    MS_STOPPING: // ---------------------------------------------------------- STOPPING MOVERS
		(*Movers are coming to a stop here in this state*)

		// Stop all movers
		allMoversHalted				:= TRUE;
		FOR i := 0 TO GVL.NUM_MOVERS - 1 DO
			Mover[i].AxisReference.ReadStatus();
			IF Mover[i].AxisReference.Status.Moving THEN
				allMoversHalted		:= FALSE;
			END_IF
		END_FOR

		GVL.XTS.Cmd.Start			:= FALSE;
 
		IF allMoversHalted THEN
           	GVL.XTS.Sts.State 		:= MS_STOPPED;
		END_IF

    MS_STOPPED: // ------------------------------------------------------------ Stop Command has been sent, hold here
		(*Movers are now stopped, and further Main Commands can be issued to the system*)

        IF GVL.XTS.Cmd.Disable THEN
            GVL.XTS.Cmd.Enable 	:= FALSE;
			GVL.XTS.Cmd.Start	:= FALSE;
            GVL.XTS.Sts.State   := MS_ONESHOT_DISABLE;
        ELSIF GVL.XTS.Cmd.Start THEN
            GVL.XTS.Cmd.Stop 	:= FALSE;
            GVL.XTS.Sts.State   := MS_ENABLING_MOVERS;
        END_IF

        // Unregister everything from everything
        FOR i := 0 TO GVL.NUM_STATIONS - 1 DO	 									Station[i].UnregisterAll();  END_FOR
		FOR i := 0 TO GVL.NUM_MULTISTATIONS - 1 DO									MultiStation[i].UnregisterAll();	END_FOR
//      FOR i := 0 TO SIZEOF(PositionTrigger) / SIZEOF(PositionTrigger[0]) - 1 DO	PositionTrigger[i].UnregisterAll();	END_FOR
//      FOR i := 0 TO SIZEOF(SpeedTrigger) / SIZEOF(SpeedTrigger[0]) - 1 DO 		SpeedTrigger[i].UnregisterAll(); END_FOR
        FOR i := 0 TO SIZEOF(Zone) / SIZEOF(Zone[0]) - 1 DO 						Zone[i].UnregisterAll();	END_FOR

	MS_ONESHOT_DISABLE:	// ------------------------------------------------------- SINGLE CYCLE ISSUE DISABLE COMMANDS
		(*Mover disable commands are issued here, followed by a state tranisition to await completion of the Disabling*)
		FOR i := 0 TO GVL.NUM_MOVERS DO
			Mover[i].Disable();
		END_FOR

		GVL.XTS.Sts.State	:=	MS_DISABLING;

    MS_DISABLING: // --------------------------------------------------- DISABLING MOVERS
		(*Movers are Disabling. During this step, we also Unregister movers from relevant Objectives
		to ensure proper startup behavior*)

        // Unregister everything from everything
        FOR i := 0 TO GVL.NUM_STATIONS - 1 DO	 									Station[i].UnregisterAll();  END_FOR
		FOR i := 0 TO GVL.NUM_MULTISTATIONS - 1 DO									MultiStation[i].UnregisterAll();	END_FOR
//      FOR i := 0 TO SIZEOF(PositionTrigger) / SIZEOF(PositionTrigger[0]) - 1 DO	PositionTrigger[i].UnregisterAll();	END_FOR
//      FOR i := 0 TO SIZEOF(SpeedTrigger) / SIZEOF(SpeedTrigger[0]) - 1 DO 		SpeedTrigger[i].UnregisterAll(); END_FOR
        FOR i := 0 TO SIZEOF(Zone) / SIZEOF(Zone[0]) - 1 DO 						Zone[i].UnregisterAll();	END_FOR
		allMoversDisabled	:= TRUE;

		FOR i := 0 TO gvl.NUM_MOVERS-1 DO
			IF NOT Mover[i].AxisReference.Status.Disabled THEN 
				allMoversDisabled	:= FALSE;
			END_IF
		END_FOR
 
        IF allMoversDisabled THEN
            GVL.XTS.Sts.State		:= MS_DISABLED;
        END_IF

    MS_ERROR: // --------------------------------------------------- ERRORSTATE
		(*A reset command can be included here to clear Mover errors, etc. and return
		to a controlled state*)

    MS_DEBUG: // ------------------------------------------------------- DEV USE ONLY
		(*This state is intentionally left blank, 
		for optional use by a developer during programming*)

END_CASE;

GVL.XTS.Sts.Enabled	:= GVL.XTS.Sts.State = MS_RUN;

// Station Actions
ACT_Orient();
ACT_BallSeat();
ACT_Print();
ACT_Vision();
ACT_Kickout();
ACT_TRAYLOAD();
ACT_IOSim();

ACT_HMIHelper();

// Initialize and update diagnostic features
InitializeUtilityLibrary();

// Call all mover function blocks cyclically
FOR i := 0 TO GVL.NUM_MOVERS - 1 DO
    Mover[i].Cyclic(GroupRef);
	Mover[i].AxisReference.ReadStatus();
END_FOR;

// Call all station function blocks cyclically
FOR i := 0 TO GVL.NUM_STATIONS - 1 DO
    Station[i].Cyclic();
END_FOR

FOR i := 0 TO GVL.NUM_MULTISTATIONS - 1 DO
	MultiStation[i].Cyclic();
END_FOR

ACTION ACT_BallSeat:
// INIT
BallSeatStation.rStation		REF= Station[GVL.STN_BALLSEAT];
BallSeatStation.rIO				REF= IO.BallSeat;
BallSeatStation.rPrintStation	REF= MultiStation[GVL.MULTISTN_PRINT];
BallSeatStation.rJobIF			REF= GVL.Job.BallSeat;

// Inputs
BallSeatStation.Enable	:= GVL.XTS.Cmd.Enable;

// FB CALLS
BallSeatStation();
END_ACTION

ACTION ACT_HMIHelper:
FOR i := 0 TO gvl.NUM_MOVERS - 1 DO
	Payload	:= Mover[i].Payload;
	HMIXTSHelper.Mover[i].BallImgVisibility			:= Payload.HasBall AND NOT Payload.Reject;
	HMIXTSHelper.Mover[i].BallRejectImgVisibility	:= Payload.HasBall AND Payload.Reject;
	HMIXTSHelper.Mover[i].MoverTextVisibility		:= Payload.HasBall;
	CASE Payload.PlayerNumber OF
	1:		HMIXTSHelper.Mover[i].MoverText		:= '1';
	2:		HMIXTSHelper.Mover[i].MoverText		:= '2';
	3:		HMIXTSHelper.Mover[i].MoverText		:= '3';
	4:		HMIXTSHelper.Mover[i].MoverText		:= '4';
	ELSE	HMIXTSHelper.Mover[i].MoverText		:= 'InvalidText';
	END_CASE
END_FOR
END_ACTION

ACTION ACT_IOSim:
// Orient
SimTimers.TON_Orient_OpenBallClamp(IN := IO.Orient.Outputs.BallClampOpen AND NOT IO.Orient.Outputs.BallClampClose, PT := T#150MS);
SimTimers.TON_Orient_CloseBallClamp(IN := IO.Orient.Outputs.BallClampClose AND NOT IO.Orient.Outputs.BallClampOpen, PT := T#150MS);
SimTimers.TON_Orient_LoadBall(IN := IO.Orient.Outputs.LoadBall, PT := T#700MS);

IF SimTimers.TON_Orient_CloseBallClamp.Q THEN		IO.Orient.Inputs.BallClampClosed	:= TRUE;	IO.Orient.Inputs.BallClampOpened	:= FALSE;	END_IF
IF SimTimers.TON_Orient_OpenBallClamp.Q THEN		IO.Orient.Inputs.BallClampOpened	:= TRUE;	IO.Orient.Inputs.BallClampClosed	:= FALSE;	END_IF
IO.Orient.Inputs.BallLoadComplete					:= SimTimers.TON_Orient_LoadBall.Q;

// Ball Seater
SimTimers.TON_BallSeat_OpenBallClamp(IN := IO.BallSeat.Outputs.BallClampOpen AND NOT IO.BallSeat.Outputs.BallClampClose, PT := T#150MS);
SimTimers.TON_BallSeat_CloseBallClamp(IN := IO.BallSeat.Outputs.BallClampClose AND NOT IO.BallSeat.Outputs.BallClampOpen, PT := T#150MS);
SimTimers.TON_BallSeat_ExtendBallSeater(IN := IO.BallSeat.Outputs.ExtendBallSeater AND NOT IO.BallSeat.Outputs.RetractBallSeater, PT := T#150MS);
SimTimers.TON_BallSeat_RetractBallSeater(IN := IO.BallSeat.Outputs.RetractBallSeater AND NOT IO.BallSeat.Outputs.ExtendBallSeater, PT := T#150MS);

IF SimTimers.TON_BallSeat_CloseBallClamp.Q THEN		IO.BallSeat.Inputs.BallClampClosed		:= TRUE;	IO.BallSeat.Inputs.BallClampOpened		:= FALSE;	END_IF
IF SimTimers.TON_BallSeat_OpenBallClamp.Q THEN		IO.BallSeat.Inputs.BallClampOpened		:= TRUE;	IO.BallSeat.Inputs.BallClampClosed		:= FALSE;	END_IF
IF SimTimers.TON_BallSeat_ExtendBallSeater.Q THEN	IO.BallSeat.Inputs.BallSeatExtended		:= TRUE;	IO.BallSeat.Inputs.BallSeatRetracted	:= FALSE;	END_IF
IF SimTimers.TON_BallSeat_RetractBallSeater.Q THEN	IO.BallSeat.Inputs.BallSeatRetracted	:= TRUE;	IO.BallSeat.Inputs.BallSeatExtended		:= FALSE;	END_IF

// Printer
SimTimers.TON_Print_PrintComplete(IN := IO.Print.Outputs.Print, PT := T#1200MS);
IO.Print.Inputs.PrintActive		:= SimTimers.TON_Print_PrintComplete.IN AND NOT SimTimers.TON_Print_PrintComplete.Q;
IO.Print.Inputs.PrintComplete	:= SimTimers.TON_Print_PrintComplete.Q;

// Vision
SimTimers.TON_Vision_ScanBall(IN := IO.Vision.Outputs.Inspect, PT := T#1000MS);
IO.Vision.Inputs.VisionActive := IO.Vision.Outputs.Inspect AND NOT(SimTimers.TON_Vision_ScanBall.Q);
IF SimTimers.TON_Vision_ScanBall.Q THEN
	IF NOT VisionComplete THEN
		VisionComplete	:= TRUE;
		IF VisTestCnt >= 9 THEN		IO.Vision.Inputs.VisionPass	:= FALSE;	IO.Vision.Inputs.VisionFail	:= TRUE;	VisTestCnt := 0;
		ELSE						IO.Vision.Inputs.VisionPass := TRUE;	IO.Vision.Inputs.VisionFail	:= FALSE;	VisTestCnt := VisTestCnt+1;
		END_IF
	END_IF
ELSE IO.Vision.Inputs.VisionPass := FALSE;	IO.Vision.Inputs.VisionFail	:= FALSE;	VisionComplete	:= FALSE;
END_IF;

// Kickout
SimTimers.TON_Kickout_OpenBallClamp(IN := IO.Kickout.Outputs.BallClampOpen AND NOT IO.Kickout.Outputs.BallClampClose, PT := T#150MS);
SimTimers.TON_Kickout_CloseBallClamp(IN := IO.Kickout.Outputs.BallClampClose AND NOT IO.Kickout.Outputs.BallClampOpen, PT := T#150MS);
SimTimers.TON_Kickout_RemoveBall(IN := IO.Kickout.Outputs.RemoveBall, PT := T#700MS);

IF SimTimers.TON_Kickout_OpenBallClamp.Q THEN		IO.Kickout.Inputs.BallClampOpened		:= TRUE;	IO.Kickout.Inputs.BallClampClosed		:= FALSE;	END_IF
IF SimTimers.TON_Kickout_CloseBallClamp.Q THEN		IO.Kickout.Inputs.BallClampClosed		:= TRUE;	IO.Kickout.Inputs.BallClampOpened		:= FALSE;	END_IF
IO.Kickout.Inputs.BallRemoved						:= SimTimers.TON_Kickout_RemoveBall.Q;

// Tray Load
SimTimers.TON_TrayLoad_OpenBallClamp(IN := IO.TrayLoad.Outputs.BallClampOpen AND NOT IO.TrayLoad.Outputs.BallClampClose, PT := T#150MS);
SimTimers.TON_TrayLoad_CloseBallClamp(IN := IO.TrayLoad.Outputs.BallClampClose AND NOT IO.TrayLoad.Outputs.BallClampOpen, PT := T#150MS);
SimTimers.TON_TrayLoad_Complete(IN := IO.TrayLoad.Outputs.LoadTray, PT := T#1500MS);

IF SimTimers.TON_TrayLoad_OpenBallClamp.Q THEN		IO.TrayLoad.Inputs.BallClampOpened		:= TRUE;	IO.TrayLoad.Inputs.BallClampClosed		:= FALSE;	END_IF
IF SimTimers.TON_TrayLoad_CloseBallClamp.Q THEN		IO.TrayLoad.Inputs.BallClampClosed		:= TRUE;	IO.TrayLoad.Inputs.BallClampOpened		:= FALSE;	END_IF
IO.TrayLoad.Inputs.TrayLoadComplete					:= SimTimers.TON_TrayLoad_Complete.Q;
END_ACTION

ACTION ACT_Kickout:
// INIT
KickoutStation.rStation			REF= Station[GVL.STN_KICKOUT];
KickoutStation.rIO				REF= IO.Kickout;
KickoutStation.rOrientStation	REF= Station[GVL.STN_ORIENT];
KickoutStation.rTrayLoadStation REF= MultiStation[GVL.MULTISTN_TRAYLOAD];
KickoutStation.rJobIF			REF= GVL.Job.Kickout;

// Inputs
KickoutStation.Enable	:= GVL.XTS.Cmd.Enable;

// FB CALLS
KickoutStation();
END_ACTION

ACTION ACT_Orient:
// INIT
OrientStation.rStation		REF= Station[GVL.STN_ORIENT];
OrientStation.rIO			REF= IO.Orient;
OrientStation.rBallSeatStn	REF= Station[GVL.STN_BALLSEAT];
OrientStation.rKickoutStn	REF= Station[GVL.STN_KICKOUT];
OrientStation.rJobIF		REF= GVL.Job.Orient;

// Inputs
OrientStation.Enable	:= GVL.XTS.Cmd.Enable;

// FB CALLS
OrientStation();
END_ACTION

ACTION ACT_Print:
// INIT
PrintStation.rMultiStn			REF= MultiStation[GVL.MULTISTN_PRINT];
PrintStation.rIO				REF= IO.Print;
PrintStation.rVisionStation		REF= Station[GVL.STN_VISION];
PrintStation.rKickoutStation	REF= Station[GVL.STN_KICKOUT];
PrintStation.rJobIF				REF= GVL.Job.Print;

// Inputs
PrintStation.Enable		:= GVL.XTS.Cmd.Enable;
PrintStation.NumColor	:= 2;
PrintStation.NumIndex	:= 2;

// FB CALLS
PrintStation();
END_ACTION

ACTION ACT_TrayLoad:
// INIT
TrayLoadStation.rMultiStn		REF= MultiStation[GVL.MULTISTN_TRAYLOAD];
TrayLoadStation.rIO				REF= IO.TrayLoad;
TrayLoadStation.rOrientStation	REF= Station[GVL.STN_ORIENT];
TrayLoadStation.rJobIF			REF= GVL.Job.TrayLoad;

// Inputs
TrayLoadStation.Enable		:= GVL.XTS.Cmd.Enable;

// FB CALLS
TrayLoadStation();
END_ACTION

ACTION ACT_Vision:
// INIT
VisionStation.rStation			REF= Station[GVL.STN_VISION];
VisionStation.rIO				REF= IO.Vision;
VisionStation.rKickoutStation	REF= Station[GVL.STN_KICKOUT];
VisionStation.rTrayloadStation	REF= MultiStation[GVL.MULTISTN_TRAYLOAD];
VisionStation.rJobIF			REF= GVL.Job.Vision;

// Inputs
VisionStation.Enable	:= GVL.XTS.Cmd.Enable;

// FB CALLS
VisionStation();
END_ACTION

ACTION InitializeUtilityLibrary:



CASE nEnvironmentState OF
	0:	// ----------------------------------------- Enable Init Items
	
		// Enable init Info Server if needed
		stXtsEnvironmentConfiguration.bEnableInitInfoServer		:= TRUE;
		
		// Enable init CA Group if needed
		stXtsEnvironmentConfiguration.bEnableInitCaGroup		:= TRUE;
		
		// Set configuration of XtsUtility init
		fbXtsEnvironment.P_XtsEnvironmentConfiguration			:= stXtsEnvironmentConfiguration;
		
		// Next step
		nEnvironmentState	:= 1;
		
	1:	// ------------------------------------------ Init Environment
		
		// Start init
		IF fbXtsEnvironment.Init(TRUE) THEN
			// stop init
			fbXtsEnvironment.Init(FALSE);
			
			// next step
			nEnvironmentState	:= 2;
		END_IF
		
	2:	// ------------------------------------------ Check for success
	
		// Check IsInitialized property
		IF fbXtsEnvironment.P_IsInitialized THEN
			// next step
			nEnvironmentState	:= 3;
		END_IF
		
	3:	// ------------------------------------------- Init Visu
	
		fbXtsEnvironmentVisu( ipTcIoXtsEnvironment := fbXtsEnvironment );
		
		// next step
		nEnvironmentState	:= 4;
		
	4:	// ------------------------------------------- Init done

		fbXtsEnvironmentVisu.Cycle();
		
END_CASE
END_ACTION

END_PROGRAM

// ---- POUs/XTS/BallPrinterStations/OrientStation.TcPOU
FUNCTION_BLOCK OrientStation EXTENDS MachineStation
VAR_INPUT
	rIO				: REFERENCE TO Orient_IO_typ;
	rStation		: REFERENCE TO Station;
	rBallSeatStn	: REFERENCE TO Station;
	rKickoutStn		: REFERENCE TO Station;
END_VAR
VAR_OUTPUT
END_VAR
VAR
	Payload	: Payload_typ;
	i: INT;
END_VAR

IF NOT (__ISVALIDREF(rStation) AND __ISVALIDREF(rIO) AND __ISVALIDREF(rBallSeatStn) AND __ISVALIDREF(rKickoutStn)) THEN
	ADSLOGSTR( ADSLOG_MSGTYPE_ERROR, 'Invalid reference at %s.', InstancePath);	// how to make this work?
	RETURN;
END_IF

IF Enable THEN
	IF NOT _Enable THEN
		;
	END_IF

	CASE State OF
		STN_WAIT:
			IF rJobIF.Cmd.Run AND rStation.MoverInPosition AND NOT rJobIF.Sts.Done THEN
				State	:= STN_CHECKMOVER;
				Payload	:= rStation.CurrentMover.Payload;
			END_IF

		STN_CHECKMOVER:
			IF NOT Payload.Init THEN
				Payload.Init	:= TRUE;
			END_IF

			IF rIO.Inputs.BallPresent THEN
				// DO NOTHING FOR NOW
			ELSE
				rIO.Outputs.BallClampOpen	:= TRUE;
				State						:= STN_OPENBALLCLAMP;
			END_IF

		STN_OPENBALLCLAMP:
			IF rIO.Inputs.BallClampOpened THEN
				rIO.Outputs.BallClampOpen	:= FALSE;
				rIO.Outputs.LoadBall		:= TRUE;
				State						:= STN_PROCESS;
			END_IF

		STN_PROCESS:
			IF rIO.Inputs.BallLoadComplete THEN
				rIO.Outputs.LoadBall		:= FALSE;
				Payload.HasBall				:= TRUE;
				FOR i := 0 TO 3 DO
					IF rJobIF.Sts.PlayerNumberCount[i] < rJobIF.Cmd.PlayerNumberCount[i] THEN
						Payload.PlayerNumber		:= i+1;
						EXIT;
					END_IF
				END_FOR
				rIO.Outputs.BallClampClose	:= TRUE;
				State						:= STN_CLOSEBALLCLAMP;
			END_IF

		STN_CLOSEBALLCLAMP:
			IF rIO.Inputs.BallClampClosed THEN
				rIO.Outputs.BallClampClose	:= FALSE;
				State						:= STN_SEND;
			END_IF

		STN_SEND:
			rJobIF.Sts.PlayerNumberCount[Payload.PlayerNumber - 1]	:= rJobIF.Sts.PlayerNumberCount[Payload.PlayerNumber - 1] + 1;
			rStation.CurrentMover.Payload	:= Payload;
			rStation.CurrentMover.MoveToStation(rBallSeatStn);
			rStation.UnregisterCurrent();
			State							:= STN_WAIT;
		
		STN_ERROR:
	
	END_CASE

	// Statuses
	rJobIF.Sts.Done	:= TRUE;
	FOR i := 0 TO 3 DO
		IF rJobIF.Sts.PlayerNumberCount[i] < rJobIF.Cmd.PlayerNumberCount[i] THEN
			rJobIF.Sts.Done	:= FALSE;	EXIT;
		END_IF
	END_FOR


ELSIF _Enable THEN
	rIO.Outputs.BallClampClose	:= FALSE;
	rIO.Outputs.BallClampOpen	:= FALSE;
	rIO.Outputs.LoadBall		:= FALSE;
	State	:= STN_WAIT;
END_IF

//Save Previous Values
_Enable	:= Enable;

END_FUNCTION_BLOCK

// ---- POUs/XTS/BallPrinterStations/MachineStation.TcPOU
FUNCTION_BLOCK MachineStation
VAR_INPUT
	Enable	: BOOL;
	Run		: BOOL;
	Reset	: BOOL;
	rJobIF			: REFERENCE TO JobStn_typ;
END_VAR
VAR_OUTPUT
	State	: StnState_Enum;
	Error	: BOOL;
	ErrorID	: DINT;
END_VAR
VAR
	_Enable	: BOOL;

    {attribute 'instance-path'}
    {attribute 'noinit'}
    InstancePath 				: STRING; // Unique variable path of the instance
END_VAR

END_FUNCTION_BLOCK

// ---- POUs/XTS/BallPrinterStations/BallSeatStation.TcPOU
FUNCTION_BLOCK BallSeatStation EXTENDS MachineStation
VAR_INPUT
	rIO				: REFERENCE TO BallSeat_IO_typ;
	rStation		: REFERENCE TO Station;
	rPrintStation	: REFERENCE TO MultiStation;
END_VAR
VAR_OUTPUT
END_VAR
VAR
	Payload	: Payload_typ;
END_VAR

IF NOT (__ISVALIDREF(rStation) AND __ISVALIDREF(rIO) AND __ISVALIDREF(rPrintStation)) THEN
	ADSLOGSTR( ADSLOG_MSGTYPE_ERROR, 'Invalid reference at %s.', InstancePath);	// how to make this work?
	RETURN;
END_IF

// WHATS THE DIFFERENCE BETWEEN PUTTING THIS HERE VS FB.Cyclic Method?

IF Enable THEN
	IF NOT _Enable THEN
		;
	END_IF

	CASE State OF
		STN_WAIT:
			IF rJobIF.Cmd.Run AND rStation.MoverInPosition THEN
				Payload						:= rStation.CurrentMover.Payload;
				rIO.Outputs.BallClampOpen	:= TRUE;
				State						:= STN_OPENBALLCLAMP;
			END_IF

		STN_OPENBALLCLAMP:
			IF rIO.Inputs.BallClampOpened THEN
				rIO.Outputs.BallClampOpen		:= FALSE;
				rIO.Outputs.ExtendBallSeater	:= TRUE;
				State							:= STN_PROCESS;
			END_IF

		STN_PROCESS:
			IF rIO.Inputs.BallSeatExtended THEN
				rIO.Outputs.ExtendBallSeater	:= FALSE;
				rIO.Outputs.RetractBallSeater	:= TRUE;
				Payload.BallSeated				:= TRUE;
				rIO.Outputs.BallClampClose		:= TRUE;
				State							:= STN_CLOSEBALLCLAMP;
			END_IF

		STN_CLOSEBALLCLAMP:
			IF rIO.Inputs.BallClampClosed AND rIO.Inputs.BallSeatRetracted THEN
				rIO.Outputs.RetractBallSeater	:= FALSE;
				rIO.Outputs.BallClampClose		:= FALSE;
				State							:= STN_SEND;
			END_IF

		STN_SEND:
			rStation.CurrentMover.Payload	:= Payload;
			rStation.CurrentMover.MoveToMultiStation(rPrintStation);
			rStation.UnregisterCurrent();
			State							:= STN_WAIT;
		
		STN_ERROR:
	
	END_CASE

ELSIF _Enable THEN
	rIO.Outputs.BallClampClose		:= FALSE;
	rIO.Outputs.BallClampOpen		:= FALSE;
	rIO.Outputs.ExtendBallSeater	:= FALSE;
	rIO.Outputs.RetractBallSeater	:= FALSE;
	State	:= STN_WAIT;
END_IF

//Save Previous Values
_Enable	:= Enable;

END_FUNCTION_BLOCK

// ---- POUs/XTS/BallPrinterStations/PrintStation.TcPOU
FUNCTION_BLOCK PrintStation EXTENDS MachineStation
VAR_INPUT
	rIO				: REFERENCE TO Print_IO_typ;
	rMultiStn		: REFERENCE TO MultiStation;
	rVisionStation	: REFERENCE TO Station;
	rKickoutStation	: REFERENCE TO Station;
	NumIndex		: USINT;
	NumColor		: USINT;
END_VAR
VAR_OUTPUT
END_VAR
VAR
	PosTriggerPayload	: Payload_typ;
	StationPayload		: ARRAY[0..GVL.MULTISTN_NUM_STN - 1] OF Payload_typ;
	MoverHalted			: BOOL;
	PrintConfig			: PrintConfig_typ;
	i					: INT;
	FarthestIndex0StnTrackedMovers: INT;
END_VAR

IF NOT (__ISVALIDREF(rMultiStn) AND __ISVALIDREF(rIO) AND __ISVALIDREF(rVisionStation) AND __ISVALIDREF(rKickoutStation)) THEN
	ADSLOGSTR( ADSLOG_MSGTYPE_ERROR, 'Invalid reference at %s.', InstancePath);	// how to make this work?
	RETURN;
END_IF

// Station Sequence
IF Enable THEN
	IF NOT _Enable THEN
		ACT_ConfigurePrint();
	END_IF

	// Catch Incoming Shuttles and process them
	IF rMultiStn.PositionTrigger.MoverPassedPosition THEN
(*		PosTriggerPayload	:= rMultiStn.PositionTrigger.CurrentMover.Payload;
		// Mover payload not valid for printing
		IF PosTriggerPayload.Reject OR NOT(PosTriggerPayload.HasBall AND PosTriggerPayload.BallSeated) THEN		
			PosTriggerPayload.Reject	:= TRUE;
			IF rMultiStn.TrackedMoverCount > 0 THEN
				MoverHalted				:= TRUE;
				rMultiStn.PositionTrigger.CurrentMover.Halt();
			ELSE
				rMultiStn.PositionTrigger.CurrentMover.MoveToStation(rKickoutStation);
				rMultiStn.PositionTrigger.CurrentMover.Payload	:= PosTriggerPayload;
				rMultiStn.PositionTrigger.MuteCurrent();
				MoverHalted				:= FALSE;
			END_IF
		// mover ok to print
		ELSE						*) // This doesn't work and it's not really necessary.  
										// PositionTrigger would need to buffer events.  
										// this only works when movers are going slow
										// Peter eventually going to add event buffering to position trigger, not worth doing for demo
			FarthestIndex0StnTrackedMovers	:= 100;
			FOR i := PrintConfig.LastProcessIndex0StnIndex TO 0 BY -1 DO
				IF rMultiStn.Station[i].TrackedMoverCount < FarthestIndex0StnTrackedMovers THEN
					FarthestIndex0StnTrackedMovers	:= i;
				END_IF
			END_FOR
					
			FOR i := PrintConfig.LastProcessIndex0StnIndex TO 0 BY -1 DO
				IF PrintConfig.StationEnable[i] AND PrintConfig.ProcessIndex[i] = 0 AND rMultiStn.Station[i].TrackedMoverCount = 0 THEN
					rMultiStn.PositionTrigger.CurrentMover.MoveToStation(rMultiStn.Station[i]);
					rMultiStn.PositionTrigger.MuteCurrent();
					EXIT;
				ELSIF i = 0 THEN
					rMultiStn.PositionTrigger.CurrentMover.MoveToStation(rMultiStn.Station[FarthestIndex0StnTrackedMovers]);
					rMultiStn.PositionTrigger.MuteCurrent();
					EXIT;
				END_IF
			END_FOR
		(*END_IF*)
	END_IF

	// Printing Sequence State Machine
	CASE State OF
		STN_WAIT:
			IF rJobIF.Cmd.Run AND_THEN THIS^.MoversReadyForCycle() THEN
				FOR i := 0 TO GVL.MULTISTN_NUM_STN - 1 DO
					IF rMultiStn.Station[i].TrackedMoverCount > 0 THEN
						StationPayload[i]	:= rMultiStn.Station[i].CurrentMover.Payload;
					END_IF
				END_FOR
				rIO.Outputs.Print	:= TRUE;
				State				:= STN_PROCESS;
			END_IF

		STN_PROCESS:
			IF rIO.Inputs.PrintComplete THEN
				rIO.Outputs.Print		:= FALSE;
				FOR i := 0 TO GVL.MULTISTN_NUM_STN - 1 DO
					IF rMultiStn.Station[i].TrackedMoverCount > 0 THEN
						StationPayload[i].PrintStepComplete[PrintConfig.ProcessIndex[i]]	:= TRUE;
						IF PrintConfig.FinalPrint[i] THEN 
							StationPayload[i].PrintComplete		:= TRUE;
							IF StationPayload[i].HasBall THEN
								rJobIF.Sts.PlayerNumberCount[StationPayload[i].PlayerNumber - 1] := rJobIF.Sts.PlayerNumberCount[StationPayload[i].PlayerNumber - 1] + 1;
							END_IF
						END_IF
					END_IF
				END_FOR
			State	:= STN_SEND;
			END_IF

		STN_SEND:

			// Write Payload Data
			FOR i := 0 TO GVL.MULTISTN_NUM_STN - 1 DO
				IF rMultiStn.Station[i].TrackedMoverCount > 0 THEN
					rMultiStn.Station[i].CurrentMover.Payload							:= StationPayload[i];
				END_IF
			END_FOR

			// Send Mover
			ACT_PrintSendMover();
			State	:= STN_WAIT;

		STN_ERROR:

	END_CASE

ELSIF _Enable THEN
	State	:= STN_WAIT;
END_IF

//Save Previous Values
_Enable	:= Enable;

ACTION ACT_ConfigurePrint:
memset(ADR(PrintConfig), 0, SIZEOF(PrintConfig));

CASE NumColor OF
1:
	CASE NumIndex OF
	1:	PrintConfig.StationEnable[2] := TRUE;	PrintConfig.ProcessIndex[2] := 0; PrintConfig.FinalPrint[2] := TRUE;	PrintConfig.LastProcessIndex0StnIndex	:= 2;

	2:	PrintConfig.StationEnable[1] := TRUE;	PrintConfig.ProcessIndex[1] := 0; PrintConfig.FinalPrint[1] := TRUE;
		PrintConfig.StationEnable[2] := TRUE;	PrintConfig.ProcessIndex[2] := 0; PrintConfig.FinalPrint[2] := TRUE;	PrintConfig.LastProcessIndex0StnIndex	:= 2;

	3:	PrintConfig.StationEnable[1] := TRUE;	PrintConfig.ProcessIndex[1] := 0; PrintConfig.FinalPrint[1] := TRUE;
		PrintConfig.StationEnable[2] := TRUE;	PrintConfig.ProcessIndex[2] := 0; PrintConfig.FinalPrint[2] := TRUE;
		PrintConfig.StationEnable[3] := TRUE;	PrintConfig.ProcessIndex[3] := 0; PrintConfig.FinalPrint[3] := TRUE;	PrintConfig.LastProcessIndex0StnIndex	:= 3;

	4:	PrintConfig.StationEnable[0] := TRUE;	PrintConfig.ProcessIndex[0] := 0; PrintConfig.FinalPrint[0] := TRUE;
		PrintConfig.StationEnable[1] := TRUE;	PrintConfig.ProcessIndex[1] := 0; PrintConfig.FinalPrint[1] := TRUE;
		PrintConfig.StationEnable[2] := TRUE;	PrintConfig.ProcessIndex[2] := 0; PrintConfig.FinalPrint[2] := TRUE;
		PrintConfig.StationEnable[3] := TRUE;	PrintConfig.ProcessIndex[3] := 0; PrintConfig.FinalPrint[3] := TRUE;	PrintConfig.LastProcessIndex0StnIndex	:= 3;
	END_CASE
2:
	CASE NumIndex OF
	1:	PrintConfig.StationEnable[1] := TRUE;	PrintConfig.ProcessIndex[1] := 0; PrintConfig.FinalPrint[1] := FALSE;	PrintConfig.LastProcessIndex0StnIndex	:= 1;
		PrintConfig.StationEnable[2] := TRUE;	PrintConfig.ProcessIndex[2] := 1; PrintConfig.FinalPrint[2] := TRUE;

	2:	PrintConfig.StationEnable[0] := TRUE;	PrintConfig.ProcessIndex[0] := 0; PrintConfig.FinalPrint[0] := FALSE;
		PrintConfig.StationEnable[1] := TRUE;	PrintConfig.ProcessIndex[1] := 0; PrintConfig.FinalPrint[1] := FALSE;	PrintConfig.LastProcessIndex0StnIndex	:= 1;
		PrintConfig.StationEnable[2] := TRUE;	PrintConfig.ProcessIndex[2] := 1; PrintConfig.FinalPrint[2] := TRUE;
		PrintConfig.StationEnable[3] := TRUE;	PrintConfig.ProcessIndex[3] := 1; PrintConfig.FinalPrint[3] := TRUE;
	END_CASE
3:
		PrintConfig.StationEnable[1] := TRUE;	PrintConfig.ProcessIndex[1] := 0; PrintConfig.FinalPrint[1] := FALSE;	PrintConfig.LastProcessIndex0StnIndex	:= 1;
		PrintConfig.StationEnable[2] := TRUE;	PrintConfig.ProcessIndex[2] := 1; PrintConfig.FinalPrint[2] := FALSE;
		PrintConfig.StationEnable[3] := TRUE;	PrintConfig.ProcessIndex[3] := 2; PrintConfig.FinalPrint[3] := TRUE;

4:		PrintConfig.StationEnable[0] := TRUE;	PrintConfig.ProcessIndex[0] := 0; PrintConfig.FinalPrint[0] := FALSE;	PrintConfig.LastProcessIndex0StnIndex	:= 0;
		PrintConfig.StationEnable[1] := TRUE;	PrintConfig.ProcessIndex[1] := 1; PrintConfig.FinalPrint[1] := FALSE;
		PrintConfig.StationEnable[2] := TRUE;	PrintConfig.ProcessIndex[2] := 2; PrintConfig.FinalPrint[2] := FALSE;
		PrintConfig.StationEnable[3] := TRUE;	PrintConfig.ProcessIndex[3] := 3; PrintConfig.FinalPrint[3] := TRUE;
END_CASE
END_ACTION

ACTION ACT_PrintSendMover:
CASE NumColor OF
1:
	CASE NumIndex OF
	1:	IF rMultiStn.Station[2].TrackedMoverCount > 0 THEN rMultiStn.Station[2].CurrentMover.MoveToStation(rVisionStation);			rMultiStn.Station[2].UnregisterCurrent();	END_IF

	2:	IF rMultiStn.Station[2].TrackedMoverCount > 0 THEN rMultiStn.Station[2].CurrentMover.MoveToStation(rVisionStation);			rMultiStn.Station[2].UnregisterCurrent();	END_IF
		IF rMultiStn.Station[1].TrackedMoverCount > 0 THEN rMultiStn.Station[1].CurrentMover.MoveToStation(rVisionStation);			rMultiStn.Station[1].UnregisterCurrent();	END_IF

	3:	IF rMultiStn.Station[3].TrackedMoverCount > 0 THEN rMultiStn.Station[3].CurrentMover.MoveToStation(rVisionStation);			rMultiStn.Station[3].UnregisterCurrent();	END_IF
		IF rMultiStn.Station[2].TrackedMoverCount > 0 THEN rMultiStn.Station[2].CurrentMover.MoveToStation(rVisionStation);			rMultiStn.Station[2].UnregisterCurrent();	END_IF
		IF rMultiStn.Station[1].TrackedMoverCount > 0 THEN rMultiStn.Station[1].CurrentMover.MoveToStation(rVisionStation);			rMultiStn.Station[1].UnregisterCurrent();	END_IF

	4:	IF rMultiStn.Station[3].TrackedMoverCount > 0 THEN rMultiStn.Station[3].CurrentMover.MoveToStation(rVisionStation);			rMultiStn.Station[3].UnregisterCurrent();	END_IF
		IF rMultiStn.Station[2].TrackedMoverCount > 0 THEN rMultiStn.Station[2].CurrentMover.MoveToStation(rVisionStation);			rMultiStn.Station[2].UnregisterCurrent();	END_IF
		IF rMultiStn.Station[1].TrackedMoverCount > 0 THEN rMultiStn.Station[1].CurrentMover.MoveToStation(rVisionStation);			rMultiStn.Station[1].UnregisterCurrent();	END_IF
		IF rMultiStn.Station[0].TrackedMoverCount > 0 THEN rMultiStn.Station[0].CurrentMover.MoveToStation(rVisionStation);			rMultiStn.Station[0].UnregisterCurrent();	END_IF
	END_CASE
2:
	CASE NumIndex OF
	1:	IF rMultiStn.Station[2].TrackedMoverCount > 0 THEN rMultiStn.Station[2].CurrentMover.MoveToStation(rVisionStation);			rMultiStn.Station[2].UnregisterCurrent();	END_IF
		IF rMultiStn.Station[1].TrackedMoverCount > 0 THEN rMultiStn.Station[1].CurrentMover.MoveToStation(rMultiStn.Station[2]);	rMultiStn.Station[1].UnregisterCurrent();	END_IF


	2:	IF rMultiStn.Station[3].TrackedMoverCount > 0 THEN rMultiStn.Station[3].CurrentMover.MoveToStation(rVisionStation);			rMultiStn.Station[3].UnregisterCurrent();	END_IF
		IF rMultiStn.Station[2].TrackedMoverCount > 0 THEN rMultiStn.Station[2].CurrentMover.MoveToStation(rVisionStation);			rMultiStn.Station[2].UnregisterCurrent();	END_IF
		IF rMultiStn.Station[1].TrackedMoverCount > 0 THEN rMultiStn.Station[1].CurrentMover.MoveToStation(rMultiStn.Station[3]);	rMultiStn.Station[1].UnregisterCurrent();	END_IF
		IF rMultiStn.Station[0].TrackedMoverCount > 0 THEN rMultiStn.Station[0].CurrentMover.MoveToStation(rMultiStn.Station[2]);	rMultiStn.Station[0].UnregisterCurrent();	END_IF
	END_CASE

3:		IF rMultiStn.Station[3].TrackedMoverCount > 0 THEN rMultiStn.Station[3].CurrentMover.MoveToStation(rVisionStation);			rMultiStn.Station[3].UnregisterCurrent();	END_IF
		IF rMultiStn.Station[2].TrackedMoverCount > 0 THEN rMultiStn.Station[2].CurrentMover.MoveToStation(rMultiStn.Station[3]);	rMultiStn.Station[2].UnregisterCurrent();	END_IF
		IF rMultiStn.Station[1].TrackedMoverCount > 0 THEN rMultiStn.Station[1].CurrentMover.MoveToStation(rMultiStn.Station[2]);	rMultiStn.Station[1].UnregisterCurrent();	END_IF

4:		IF rMultiStn.Station[3].TrackedMoverCount > 0 THEN rMultiStn.Station[3].CurrentMover.MoveToStation(rVisionStation);			rMultiStn.Station[3].UnregisterCurrent();	END_IF
		IF rMultiStn.Station[2].TrackedMoverCount > 0 THEN rMultiStn.Station[2].CurrentMover.MoveToStation(rMultiStn.Station[3]);	rMultiStn.Station[2].UnregisterCurrent();	END_IF
		IF rMultiStn.Station[1].TrackedMoverCount > 0 THEN rMultiStn.Station[1].CurrentMover.MoveToStation(rMultiStn.Station[2]);	rMultiStn.Station[1].UnregisterCurrent();	END_IF
		IF rMultiStn.Station[0].TrackedMoverCount > 0 THEN rMultiStn.Station[0].CurrentMover.MoveToStation(rMultiStn.Station[1]);	rMultiStn.Station[0].UnregisterCurrent();	END_IF
END_CASE
END_ACTION

ACTION ACT_PrintStatuses:

END_ACTION

METHOD MoversReadyForCycle : BOOL
// Check that all movers are in position, and that there are movers in all of the enabled process index 0 print positions
MoversReadyForCycle	:= TRUE; 
IF NOT rMultiStn.AllMoversInPosition THEN	// Any stations with tracked movers that don't have mover in position will trigger this false
	MoversReadyForCycle	:= FALSE;
ELSE
	FOR i := GVL.MULTISTN_NUM_STN - 1 TO 0 BY - 1 DO
		IF PrintConfig.StationEnable[i] AND PrintConfig.ProcessIndex[i] = 0 THEN	// Check that all process index 0 stations have movers to ensure full print cycle
			IF rMultiStn.Station[i].TrackedMoverCount = 0 AND NOT MoverHalted THEN		// Ignore this check if there is a mover halted by the position trigger
				MoversReadyForCycle	:= FALSE;
			END_IF
		END_IF
	END_FOR
END_IF
END_METHOD

END_FUNCTION_BLOCK

// ---- POUs/XTS/BallPrinterStations/VisionStation.TcPOU
FUNCTION_BLOCK VisionStation EXTENDS MachineStation
VAR_INPUT
	rIO					: REFERENCE TO Vision_IO_typ;
	rStation			: REFERENCE TO Station;
	rKickoutStation 	: REFERENCE TO Station;
	rTrayLoadStation 	: REFERENCE TO MultiStation;
END_VAR
VAR_OUTPUT
END_VAR
VAR
	Payload			: Payload_typ;
END_VAR

IF NOT (__ISVALIDREF(rStation) AND __ISVALIDREF(rIO) AND __ISVALIDREF(rKickoutStation) AND __ISVALIDREF(rTrayLoadStation)) THEN
	ADSLOGSTR( ADSLOG_MSGTYPE_ERROR, 'Invalid reference at %s.', InstancePath);	// how to make this work?
	RETURN;
END_IF

IF Enable THEN
	IF NOT _Enable THEN
		;
	END_IF

	CASE State OF
		STN_WAIT:
			IF rJobIF.Cmd.Run AND rStation.MoverInPosition THEN
				Payload	:= rStation.CurrentMover.Payload;
				IF rJobIF.Cmd.IgnoreVision THEN
					State	:= STN_SEND;
				ELSE
					State	:= STN_CHECKMOVER;
				END_IF
			END_IF

		STN_CHECKMOVER:
				
			rIO.Outputs.Inspect := TRUE; // Start inspect
			IF rIO.Inputs.VisionActive THEN
				State := STN_PROCESS;
			END_IF

		STN_PROCESS:
				IF NOT(rIO.Inputs.VisionActive)THEN
					IF rIO.Inputs.VisionPass THEN
						Payload.VisionPass 	:= TRUE;
						
					ELSIF rIO.Inputs.VisionFail THEN
						Payload.VisionPass 	:= FALSE;
						Payload.Reject		:= TRUE;
						rJobIF.Sts.RejectedPlayerNumberCount[Payload.PlayerNumber-1] := rJobIF.Sts.RejectedPlayerNumberCount[Payload.PlayerNumber-1] + 1;
						
					ELSE // Failed to get feedback. TODO: Need alarm.
					END_IF;
					
					rIO.Outputs.Inspect := FALSE;
					State 				:= STN_SEND;
				END_IF;

		STN_SEND:				
			IF Payload.Reject THEN
				rStation.CurrentMover.Payload	:= Payload;
				rStation.CurrentMover.MoveToStation(rKickoutStation);
				rStation.UnregisterCurrent();	
			ELSE
				rStation.CurrentMover.Payload	:= Payload;
				rStation.CurrentMover.MoveToMultiStation(rTrayLoadStation);
				rStation.UnregisterCurrent();
			END_IF;
			State								:= STN_WAIT;
		
		STN_ERROR:
	
	END_CASE

ELSIF _Enable THEN
	memset(ADR(rIO.Outputs), 0, SIZEOF(rIO.Outputs));
	State	:= STN_WAIT;
END_IF

//Save Previous Values
_Enable	:= Enable;

END_FUNCTION_BLOCK

// ---- POUs/XTS/BallPrinterStations/KickoutStation.TcPOU
FUNCTION_BLOCK KickoutStation EXTENDS MachineStation
VAR_INPUT
	rIO					: REFERENCE TO Kickout_IO_typ;
	rStation			: REFERENCE TO Station;
	rOrientStation 		: REFERENCE TO Station;
	rTrayLoadStation	: REFERENCE TO MultiStation;
END_VAR
VAR_OUTPUT
END_VAR
VAR
	Payload			: Payload_typ;
END_VAR

IF NOT (__ISVALIDREF(rStation) AND __ISVALIDREF(rIO) AND __ISVALIDREF(rOrientStation) ) THEN
	ADSLOGSTR( ADSLOG_MSGTYPE_ERROR, 'Invalid reference at %s.', InstancePath);	// how to make this work?
	RETURN;
END_IF

IF Enable THEN
	IF NOT _Enable THEN
		;
	END_IF

	CASE State OF
		STN_WAIT:
			IF rJobIF.Cmd.Run AND rStation.MoverInPosition THEN
				State	:= STN_CHECKMOVER;
				Payload	:= rStation.CurrentMover.Payload;
			END_IF

		STN_CHECKMOVER:
			
		IF rIO.Inputs.BallRemoved THEN 
			// Oops ??
		ELSE
			rIO.Outputs.BallClampOpen := TRUE;
			State := STN_OPENBALLCLAMP;
				
		END_IF
			
		
		STN_OPENBALLCLAMP:
			IF rIO.Inputs.BallClampOpened THEN
				rIO.Outputs.BallClampOpen	:= FALSE;
				rIO.Outputs.RemoveBall		:= TRUE;
				State						:= STN_PROCESS;
			END_IF

		STN_PROCESS:
			IF rIO.Inputs.BallRemoved THEN
				rIO.Outputs.RemoveBall		:= FALSE;
				Payload.HasBall 			:= FALSE;
				Payload.BallSeated 			:= FALSE;
				Payload.Reject 				:= FALSE;
				rIO.Outputs.BallClampClose 	:= TRUE;
				State 						:= STN_CLOSEBALLCLAMP;
			END_IF;
			
		STN_CLOSEBALLCLAMP:
			IF rIO.Inputs.BallClampClosed THEN
				rIO.Outputs.BallClampClose 	:= FALSE;
				State						:= STN_SEND;
			END_IF

		STN_SEND:

			rStation.CurrentMover.Payload	:= Payload;
			rStation.CurrentMover.MoveToMultiStation(rTrayLoadStation);
			rStation.CurrentMover.MoveToStation(rOrientStation);
			rStation.UnregisterCurrent();

			State							:= STN_WAIT;
		
		STN_ERROR:
	
	END_CASE

ELSIF _Enable THEN
	rIO.Outputs.BallClampClose	:= FALSE;
	rIO.Outputs.BallClampOpen	:= FALSE;
	rIO.Outputs.RemoveBall		:= FALSE;
	State	:= STN_WAIT;
END_IF

//Save Previous Values
_Enable	:= Enable;

END_FUNCTION_BLOCK

// ---- POUs/XTS/BallPrinterStations/TrayLoadStation.TcPOU
FUNCTION_BLOCK TrayLoadStation EXTENDS MachineStation
VAR_INPUT
	rIO				: REFERENCE TO TrayLoad_IO_typ;
	rMultiStn		: REFERENCE TO MultiStation;
	rOrientStation	: REFERENCE TO Station;
END_VAR
VAR_OUTPUT
END_VAR
VAR
	PosTriggerPayload	: Payload_typ;
	StationPayload		: ARRAY[0..GVL.MULTISTN_NUM_STN - 1] OF Payload_typ;
	MoverHalted			: BOOL;
	i					: INT;
	FarthestIndex0StnTrackedMovers: INT;
END_VAR

IF NOT (__ISVALIDREF(rMultiStn) AND __ISVALIDREF(rIO) AND __ISVALIDREF(rOrientStation)) THEN
	ADSLOGSTR( ADSLOG_MSGTYPE_ERROR, 'Invalid reference at %s.', InstancePath);	// how to make this work?
	RETURN;
END_IF

// Station Sequence
IF Enable THEN
	IF NOT _Enable THEN
		;
	END_IF

	// Catch Incoming Shuttles and process them
	IF rMultiStn.PositionTrigger.MoverPassedPosition THEN
(*		PosTriggerPayload	:= rMultiStn.PositionTrigger.CurrentMover.Payload;
		// Mover payload not valid for printing
		IF PosTriggerPayload.Reject OR NOT(PosTriggerPayload.HasBall AND PosTriggerPayload.BallSeated) THEN		
			PosTriggerPayload.Reject	:= TRUE;
			IF rMultiStn.TrackedMoverCount > 0 THEN
				MoverHalted				:= TRUE;
				rMultiStn.PositionTrigger.CurrentMover.Halt();
			ELSE
				rMultiStn.PositionTrigger.CurrentMover.MoveToStation(rKickoutStation);
				rMultiStn.PositionTrigger.CurrentMover.Payload	:= PosTriggerPayload;
				rMultiStn.PositionTrigger.MuteCurrent();
				MoverHalted				:= FALSE;
			END_IF
		// mover ok to print
		ELSE						*) // This doesn't work and it's not really necessary.  
										// PositionTrigger would need to buffer events.  
										// this only works when movers are going slow
										// Peter eventually going to add event buffering to position trigger, not worth doing for demo
			FarthestIndex0StnTrackedMovers	:= 100;
			FOR i := 3 TO 0 BY -1 DO
				IF rMultiStn.Station[i].TrackedMoverCount < FarthestIndex0StnTrackedMovers THEN
					FarthestIndex0StnTrackedMovers	:= i;
				END_IF
			END_FOR
					
			FOR i := 3 TO 0 BY -1 DO
				IF rMultiStn.Station[i].TrackedMoverCount = 0 THEN
					rMultiStn.PositionTrigger.CurrentMover.MoveToStation(rMultiStn.Station[i]);
					rMultiStn.PositionTrigger.MuteCurrent();
					EXIT;
				ELSIF i = 0 THEN
					rMultiStn.PositionTrigger.CurrentMover.MoveToStation(rMultiStn.Station[FarthestIndex0StnTrackedMovers]);
					rMultiStn.PositionTrigger.MuteCurrent();
					EXIT;
				END_IF
			END_FOR
		(*END_IF*)
	END_IF

	// Printing Sequence State Machine
	CASE State OF
		STN_WAIT:
			IF rJobIF.Cmd.Run AND_THEN THIS^.MoversReadyForCycle() THEN
				FOR i := 0 TO GVL.MULTISTN_NUM_STN - 1 DO
					IF rMultiStn.Station[i].TrackedMoverCount > 0 THEN
						StationPayload[i]	:= rMultiStn.Station[i].CurrentMover.Payload;
					END_IF
				END_FOR
				rIO.Outputs.BallClampOpen	:= TRUE;
				State						:= STN_OPENBALLCLAMP;
			END_IF

		STN_OPENBALLCLAMP:
			IF rIO.Inputs.BallClampOpened THEN
				rIO.Outputs.BallClampOpen	:= FALSE;
				rIO.Outputs.LoadTray		:= TRUE;
				State						:= STN_PROCESS;
			END_IF

		STN_PROCESS:
			IF rIO.Inputs.TrayLoadComplete THEN
				rIO.Outputs.LoadTray		:= FALSE;
				FOR i := 0 TO GVL.MULTISTN_NUM_STN - 1 DO
					IF rMultiStn.Station[i].TrackedMoverCount > 0 THEN
						IF StationPayload[i].HasBall THEN
							rJobIF.Sts.PlayerNumberCount[StationPayload[i].PlayerNumber - 1] := rJobIF.Sts.PlayerNumberCount[StationPayload[i].PlayerNumber - 1] + 1;
						END_IF
						RemoveBallFromPayload(StationPayload[i]);
					END_IF
				END_FOR
			rIO.Outputs.BallClampClose	:= TRUE;
			State						:= STN_CLOSEBALLCLAMP;
			END_IF

		STN_CLOSEBALLCLAMP:
			IF rIO.Inputs.BallClampClosed THEN
				rIO.Outputs.BallClampClose	:= FALSE;
				State						:= STN_SEND;
			END_IF

		STN_SEND:
			// Write Payload Data
			FOR i := 0 TO GVL.MULTISTN_NUM_STN - 1 DO
				IF rMultiStn.Station[i].TrackedMoverCount > 0 THEN
					rMultiStn.Station[i].CurrentMover.Payload		:= StationPayload[i];
				END_IF
			END_FOR

			// Send Mover
			ACT_TLSendMover();
			State	:= STN_WAIT;

		STN_ERROR:

	END_CASE

	// Statuses
	rJobIF.Sts.Done	:= TRUE;
	FOR i := 0 TO 3 DO
		IF rJobIF.Sts.PlayerNumberCount[i] < rJobIF.Cmd.PlayerNumberCount[i] THEN
			rJobIF.Sts.Done	:= FALSE;	EXIT;
		END_IF
	END_FOR

ELSIF _Enable THEN
	memset(ADR(rIO.Outputs), 0, SIZEOF(rIO.Outputs));
	rJobIF.Sts.Done	:= FALSE;
	State			:= STN_WAIT;
END_IF

//Save Previous Values
_Enable	:= Enable;

ACTION ACT_TLSendMover:

IF rMultiStn.Station[3].TrackedMoverCount > 0 THEN rMultiStn.Station[3].CurrentMover.MoveToStation(rOrientStation);		rMultiStn.Station[3].UnregisterCurrent();	END_IF
IF rMultiStn.Station[2].TrackedMoverCount > 0 THEN rMultiStn.Station[2].CurrentMover.MoveToStation(rOrientStation);		rMultiStn.Station[2].UnregisterCurrent();	END_IF
IF rMultiStn.Station[1].TrackedMoverCount > 0 THEN rMultiStn.Station[1].CurrentMover.MoveToStation(rOrientStation);		rMultiStn.Station[1].UnregisterCurrent();	END_IF
IF rMultiStn.Station[0].TrackedMoverCount > 0 THEN rMultiStn.Station[0].CurrentMover.MoveToStation(rOrientStation);		rMultiStn.Station[0].UnregisterCurrent();	END_IF
END_ACTION

METHOD MoversReadyForCycle : BOOL
// Check that all movers are in position, and that there are movers in all of the enabled process index 0 print positions
MoversReadyForCycle	:= TRUE; 
IF NOT rMultiStn.AllMoversInPosition THEN	// Any stations with tracked movers that don't have mover in position will trigger this false
	MoversReadyForCycle	:= FALSE;
ELSE
	FOR i := GVL.MULTISTN_NUM_STN - 1 TO 0 BY - 1 DO
		IF rMultiStn.Station[i].TrackedMoverCount = 0 AND NOT MoverHalted THEN		// Ignore this check if there is a mover halted by the position trigger
			MoversReadyForCycle	:= FALSE;
		END_IF
	END_FOR
END_IF
END_METHOD

END_FUNCTION_BLOCK

// ---- POUs/XTS/BallPrinterStations/Helpers/RemoveBallFromPayload.TcPOU
FUNCTION RemoveBallFromPayload : BOOL
VAR_INPUT
	rPayload	: REFERENCE TO Payload_typ;
END_VAR
VAR
	i			: INT;
END_VAR

rPayload.HasBall		:= FALSE;
rPayload.BallSeated		:= FALSE;
rPayload.PlayerNumber	:= 0;
rPayload.PrintComplete	:= FALSE;
FOR i := 0 TO SIZEOF(rPayload.PrintStepComplete) / SIZEOF(rPayload.PrintStepComplete[0]) - 1 DO
	rPayload.PrintStepComplete[i]	:= FALSE;
END_FOR
rPayload.Reject			:= FALSE;
rPayload.VisionPass		:= FALSE;

END_FUNCTION

// ---- POUs/JobMgr.TcPOU
FUNCTION_BLOCK JobMgr
VAR_INPUT
	Cmd:	JobCmd_typ;
	rXTS:	REFERENCE TO XTSMainControl_typ;
	rRecoveryZone: REFERENCE TO Zone;
END_VAR
VAR_OUTPUT
	Sts:		JobSts_typ;
END_VAR
VAR
	State:		JobState_enum;
	Orient:		JobStn_typ;
	BallSeat:	JobStn_typ;
	Print:		JobStn_typ;
	Vision:		JobStn_typ;
	Kickout:	JobStn_typ;
	TrayLoad:	JobStn_typ;
	System:		JobStn_typ;

	StnCmdRun:	BOOL;
	StnStsAllNotRunning: BOOL;
	Payload	: Payload_typ;

	_State:		JobState_enum;
	i: INT;
END_VAR

CASE State OF
	Job_Disabled:
		IF _State <> Job_Disabled THEN
			;//Clear Job Statuses and Counts
		END_IF

		IF Cmd.Run AND rXTS.Sts.Enabled THEN
			StnCmdRun	:= TRUE;
			State		:= Job_Running;
		END_IF

	Job_Starting:
		;

	Job_Running:
		IF Sts.Done THEN
			StnCmdRun	:= FALSE;
			State		:= Job_Done;
		ELSIF Cmd.Cleanout OR NOT Cmd.Run THEN
			StnCmdRun	:= FALSE;
			State		:= Job_Pausing;
		END_IF

	Job_Pausing:
		IF Cmd.Run THEN
			StnCmdRun	:= TRUE;
			State		:= Job_Running;
		ELSIF Cmd.Cleanout AND StnStsAllNotRunning THEN
			;//MEMSET(rjo
		END_IF

	Job_Paused:
		IF Cmd.Run THEN
			StnCmdRun	:= TRUE;
			State		:= Job_Running;
		ELSIF Cmd.Cleanout THEN
			StnCmdRun	:= FALSE;
			//Sts. 
		END_IF

	Job_Done:
		IF NOT Cmd.Run THEN
			State	:= Job_Disabled;
		END_IF

	Job_Cleanout:
		IF Sts.CleanoutDone AND NOT Cmd.Cleanout THEN
			State	:= Job_Disabled;
		END_IF
END_CASE;

// Stn Commands
Orient.Cmd.Run := BallSeat.Cmd.Run := Print.Cmd.Run := StnCmdRun := Vision.Cmd.Run := Kickout.Cmd.Run := TrayLoad.Cmd.Run := StnCmdRun;

// Stn Specific Commands
FOR i := 0 TO 3 DO
	Orient.Cmd.PlayerNumberCount[i]	:= (Cmd.PlayerNumberCount[0] * 12) + Sts.RejectedPlayerNumberCount[i];
END_FOR
Print.Cmd.NumColor		:= Cmd.NumColor;
Print.Cmd.NumIndex		:= Cmd.NumIndex;
Print.Cmd.IgnoreVision	:= Cmd.IgnoreVision;
Vision.Cmd.IgnoreVision	:= Cmd.IgnoreVision;

// Stn Statuses
StnStsAllNotRunning := NOT (Orient.Sts.Running OR BallSeat.Sts.Running OR Print.Sts.Running OR Vision.Sts.Running OR Kickout.Sts.Running OR TrayLoad.Sts.Running);

// Outputs
Sts.Running						:= State = Job_Running;
Sts.Done						:= State = Job_Done;
Sts.PlayerNumberCount			:= TrayLoad.Sts.PlayerNumberCount;
Sts.PrintedPlayerNumberCount	:= Print.Sts.PlayerNumberCount;
FOR i := 0 TO 3 DO
Sts.RejectedPlayerNumberCount[i]	:= Orient.Sts.RejectedPlayerNumberCount[i] + BallSeat.Sts.RejectedPlayerNumberCount[i] +
									Print.Sts.RejectedPlayerNumberCount[i] + Vision.Sts.RejectedPlayerNumberCount[i] +
									Kickout.Sts.RejectedPlayerNumberCount[i] + Trayload.Sts.RejectedPlayerNumberCount[i] +
									System.Sts.RejectedPlayerNumberCount[i];
END_FOR

// Save Previous Values
_State	:= State;

END_FUNCTION_BLOCK

// ---- VISUs/Controls.TcVIS
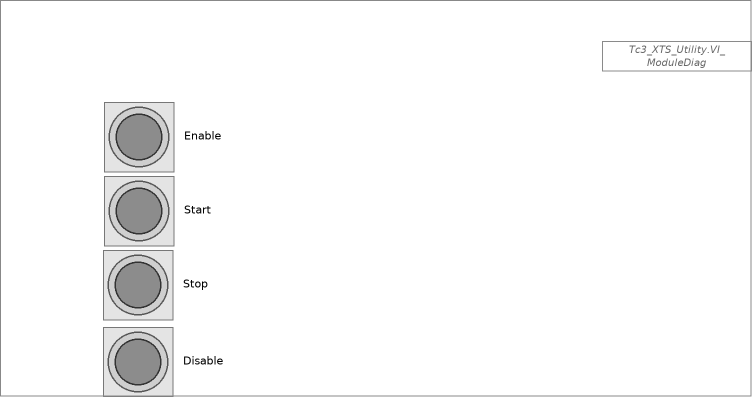
VISUALIZATION Controls  // 752x397
    PushSwitchLed (104,102 70x70), variable: GVL.XTS.Cmd.Enable, behaviour: TOGGLE, style: Switch-PushSwitchLed-Gray
    Label (181,121 150x30), "Enable"
    Label (181,195 150x30), "Start"
    PushSwitchLed (104,176 70x70), variable: GVL.XTS.Cmd.Start, behaviour: TOGGLE, style: Switch-PushSwitchLed-Gray
    Label (180,269 150x30), "Stop"
    PushSwitchLed (103,250 70x70), variable: GVL.XTS.Cmd.Stop, behaviour: TOGGLE, style: Switch-PushSwitchLed-Gray
    Label (180,346 150x30), "Disable"
    PushSwitchLed (103,327 70x70), variable: GVL.XTS.Cmd.Disable, behaviour: TOGGLE, style: Switch-PushSwitchLed-Gray
    Frame (602,41 150x30)
        shows Tc3_XTS_Utility.VI_ModuleDiag()
END_VISUALIZATION
